Universal Robots PolyScope program: Programa_UR5_Gavetas.urp

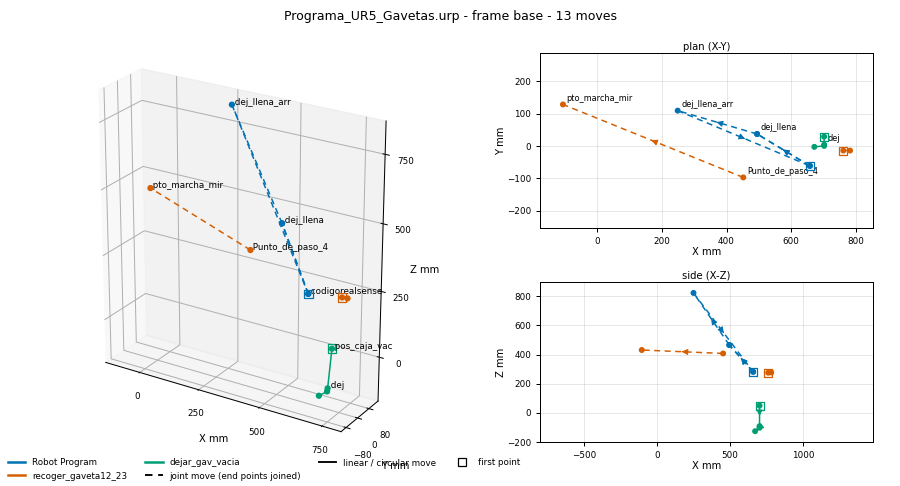
[picture p0: tool path of Programa_UR5_Gavetas.urp in frame base, 13 of 26 moves have a stored position in this frame; points joined in program order, loops and branches not executed]
Program Einnek_Planta240614 (installation=einnek directory=/programs/usbdisk/ur_mir createdIn=5.12.1.1101497 lastSavedIn=5.12.1.1101497 robotSerialNumber=20225590038)
Calibrated DH parameters: a=[0.000213, -0.400573, -0.367685, -0.000006, 0.000089, 0]; d=[0.162722, -86.393777, 65.991912, 20.535232, 0.099742, 0.099568]; alpha=[1.570328, 0.001648, 0.006729, 1.570321, -1.569293, 0]; deltaTheta=[0, -0.341442, -0.015889, 0.357341, 0.000001, 0]
InitVariablesNode variables(variable(name=ETAPA, expression=0), variable(name=IZQ_DER, expression=0), variable(name=LLENA_VACIA, expression=0), variable(name=Num_progr, expression=0), variable(name=pos_z, expression=0))
BeforeStart
  SuppressedNode
    Num_progr := 10   [initializeExpression=0]
  Folder Lectura posiciones
    URCap Read MiR register (MiRintegration, Mobile Industrial Robots APs) dataModel(register=Pos X, Variable(key=selectedVar, variable(name=pos_x, initializeExpression=0)))
    URCap Read MiR register (MiRintegration, Mobile Industrial Robots APs) dataModel(register=Pos Y, Variable(key=selectedVar, variable(name=pos_y, initializeExpression=0)))
    URCap Read MiR register (MiRintegration, Mobile Industrial Robots APs) dataModel(register=Pos Z, Variable(key=selectedVar, variable(name=pos_z, initializeExpression=0)))
    URCap Read MiR register (MiRintegration, Mobile Industrial Robots APs) dataModel(register=Rot X, Variable(key=selectedVar, variable(name=rot_x, initializeExpression=0)))
    URCap Read MiR register (MiRintegration, Mobile Industrial Robots APs) dataModel(register=Rot Y, Variable(key=selectedVar, variable(name=rot_y, initializeExpression=0)))
    URCap Read MiR register (MiRintegration, Mobile Industrial Robots APs) dataModel(register=Rot Z, Variable(key=selectedVar, variable(name=rot_z, initializeExpression=0)))
    URCap Read MiR register (MiRintegration, Mobile Industrial Robots APs) dataModel(register=IZQ_DER, Variable(key=selectedVar, variable(name=IZQ_DER, initializeExpression=0)))
    URCap Read MiR register (MiRintegration, Mobile Industrial Robots APs) dataModel(register=Altura_gaveta, Variable(key=selectedVar, variable(name=AbaArr)))
    SuppressedNode
      pos_caja := p[pos_x,pos_y,pos_z,rot_x,rot_y,rot_z]
    pos_caja := p[pos_x,pos_y,pos_z+0.12*AbaArr,rot_x,rot_y,rot_z]
  SuppressedNode
    AbaArr := 0
  SuppressedNode
    pos_caja := p[0,0,0,0,0,0]
Robot Program (runOnlyOnce=false)
  SafeHome (positionOptionType=SPEED_AND_ACCELERATION speed=1.047198 acceleration=1.396263 nextMotionTime=2)
  URCap Read MiR register (MiRintegration, Mobile Industrial Robots APs) dataModel(register=VACIA0_LLENA1, Variable(key=selectedVar, variable(name=LLENA_VACIA, initializeExpression=0)))
  If LLENA_VACIA≟1
    Folder PROGRAMA GAVETA LLENA
      URCap Read MiR register (MiRintegration, Mobile Industrial Robots APs) dataModel(register=ETAPAS, Variable(key=selectedVar, variable(name=ETAPA, initializeExpression=0)))
      Loop While (checkContinuously=false) expression=ETAPA≠101
        URCap Read MiR register (MiRintegration, Mobile Industrial Robots APs) dataModel(register=ETAPAS, Variable(key=selectedVar, variable=ETAPA))
        Wait Sleep waitTime=3
        Script: sync()
      MoveJ speed 60 deg/s, acceleration 80 deg/s^2 (useActiveTCP=true) feature=Base
        Waypoint codigorealsense: TCP in base x=657.88 y=-61.539 z=282.139 mm, rx=2.1337 ry=-2.1191 rz=-0.1759 rad; joints [160.264, -77.43, 101.576, -104.858, -93.53, -19.909] deg; TCP offset x=0 y=-115.54 z=0 mm, rx=0 ry=0 rz=0 rad
      Loop While (checkContinuously=false) expression=ETAPA≠103
        URCap Read MiR register (MiRintegration, Mobile Industrial Robots APs) dataModel(register=ETAPAS, Variable(key=selectedVar, variable=ETAPA))
        Wait Sleep waitTime=3
        Script: sync()
      Wait Sleep waitTime=1
      URCap Read MiR register (MiRintegration, Mobile Industrial Robots APs) dataModel(register=Pos_X_recogida, Variable(key=selectedVar, variable(name=PosXRecogida, initializeExpression=0)))
      Call recoger_gaveta12_23
      URCap Write MiR register (MiRintegration, Mobile Industrial Robots APs) dataModel(value=104, register=ETAPAS)
      URCap Read MiR register (MiRintegration, Mobile Industrial Robots APs) dataModel(register=ETAPAS, Variable(key=selectedVar, variable=ETAPA))
      Loop While (checkContinuously=false) expression=ETAPA≠106
        URCap Read MiR register (MiRintegration, Mobile Industrial Robots APs) dataModel(register=ETAPAS, Variable(key=selectedVar, variable=ETAPA))
        Wait Sleep waitTime=3
        Script: sync()
      Wait Condition expression=ETAPA≟106
      Folder Lectura posiciones
        URCap Read MiR register (MiRintegration, Mobile Industrial Robots APs) dataModel(register=Pos X, Variable(key=selectedVar, variable=pos_x))
        URCap Read MiR register (MiRintegration, Mobile Industrial Robots APs) dataModel(register=Pos Y, Variable(key=selectedVar, variable=pos_y))
        URCap Read MiR register (MiRintegration, Mobile Industrial Robots APs) dataModel(register=Pos Z, Variable(key=selectedVar, variable=pos_z))
        URCap Read MiR register (MiRintegration, Mobile Industrial Robots APs) dataModel(register=Rot X, Variable(key=selectedVar, variable=rot_x))
        URCap Read MiR register (MiRintegration, Mobile Industrial Robots APs) dataModel(register=Rot Y, Variable(key=selectedVar, variable=rot_y))
        URCap Read MiR register (MiRintegration, Mobile Industrial Robots APs) dataModel(register=Rot Z, Variable(key=selectedVar, variable=rot_z))
        URCap Read MiR register (MiRintegration, Mobile Industrial Robots APs) dataModel(register=IZQ_DER, Variable(key=selectedVar, variable=IZQ_DER))
        URCap Read MiR register (MiRintegration, Mobile Industrial Robots APs) dataModel(register=Altura_gaveta, Variable(key=selectedVar, variable=AbaArr))
        SuppressedNode
          pos_caja := p[pos_x,pos_y,pos_z,rot_x,rot_y,rot_z]
        SuppressedNode
          AbaArr := 0
        pos_caja := p[pos_x,pos_y,pos_z+0.12*AbaArr,rot_x,rot_y,rot_z]
      URCap Write MiR register (MiRintegration, Mobile Industrial Robots APs) dataModel(value=107, register=ETAPAS)
      If pos_z≤0.6
        MoveJ speed 60 deg/s, acceleration 80 deg/s^2 (useActiveTCP=true) feature=Base
          Waypoint dej_llena: motionParameters(jointSpeed=1.047198 jointAcceleration=0.436332 cartesianSpeed=0.25 cartesianAcceleration=1.2 blendRadius=0.05); TCP in base x=494.444 y=37.151 z=465.918 mm, rx=-2.1193 ry=2.1657 rz=-0.1543 rad; joints [165.601, -108.768, 117.243, -106.569, -87.444, -13.084] deg; TCP offset x=1.251 y=-112.953 z=-27.309 mm, rx=0 ry=0 rz=0 rad
      Else 
        MoveJ speed 60 deg/s, acceleration 80 deg/s^2 (useActiveTCP=true) feature=Base
          Waypoint dej_llena_arr: motionParameters(jointSpeed=1.047198 jointAcceleration=0.436332 cartesianSpeed=0.25 cartesianAcceleration=1.2 blendRadius=0.05); TCP in base x=248.72 y=109.415 z=823.024 mm, rx=-2.2887 ry=2.1434 rz=-0.0254 rad; joints [166.2, -111.162, 44.661, -24.388, -90.221, -17.987] deg; TCP offset x=0 y=-115.54 z=0 mm, rx=0 ry=0 rz=0 rad
      URCap Read MiR register (MiRintegration, Mobile Industrial Robots APs) dataModel(register=IZQ_DER, Variable(key=selectedVar, variable=IZQ_DER))
      If IZQ_DER≟1
        Call dejar_gav_der
      ElseIf IZQ_DER≟0
        Call dejar_gav_izq
      Else 
        Popup Message (haltProgram=false message=lado no asociado a codigo inputType=Text)
      URCap Write MiR register (MiRintegration, Mobile Industrial Robots APs) dataModel(value=108, register=ETAPAS)
      SafeHome (positionOptionType=SPEED_AND_ACCELERATION speed=1.047198 acceleration=1.396263 nextMotionTime=2)
  ElseIf LLENA_VACIA≟0
    Folder PROGRAMA GAVETA VACIA
      URCap Read MiR register (MiRintegration, Mobile Industrial Robots APs) dataModel(register=ETAPAS, Variable(key=selectedVar, variable=ETAPA))
      Loop While (checkContinuously=false) expression=ETAPA≠201
        URCap Read MiR register (MiRintegration, Mobile Industrial Robots APs) dataModel(register=ETAPAS, Variable(key=selectedVar, variable=ETAPA))
        Wait Sleep waitTime=3
        Script: sync()
      MoveJ speed 60 deg/s, acceleration 80 deg/s^2 (useActiveTCP=true) feature=Base
        Waypoint codigorealsense: TCP in base x=657.88 y=-61.539 z=282.139 mm, rx=2.1337 ry=-2.1191 rz=-0.1759 rad; joints [160.264, -77.43, 101.576, -104.858, -93.53, -19.909] deg
      Loop While (checkContinuously=false) expression=ETAPA≠203
        URCap Read MiR register (MiRintegration, Mobile Industrial Robots APs) dataModel(register=ETAPAS, Variable(key=selectedVar, variable=ETAPA))
        Wait Sleep waitTime=3
        Script: sync()
      Wait Condition expression=ETAPA≟203
      URCap Read MiR register (MiRintegration, Mobile Industrial Robots APs) dataModel(register=Pos_X_recogida, Variable(key=selectedVar, variable=PosXRecogida))
      Call recoger_gaveta12_23
      URCap Write MiR register (MiRintegration, Mobile Industrial Robots APs) dataModel(value=204, register=ETAPAS)
      SuppressedNode
        Folder Lectura posiciones
          URCap Read MiR register (MiRintegration, Mobile Industrial Robots APs) dataModel(register=Pos X, Variable(key=selectedVar, variable=pos_x))
          URCap Read MiR register (MiRintegration, Mobile Industrial Robots APs) dataModel(register=Pos Y, Variable(key=selectedVar, variable=pos_y))
          URCap Read MiR register (MiRintegration, Mobile Industrial Robots APs) dataModel(register=Pos Z, Variable(key=selectedVar, variable=pos_z))
          URCap Read MiR register (MiRintegration, Mobile Industrial Robots APs) dataModel(register=Rot X, Variable(key=selectedVar, variable=rot_x))
          URCap Read MiR register (MiRintegration, Mobile Industrial Robots APs) dataModel(register=Rot Y, Variable(key=selectedVar, variable=rot_y))
          URCap Read MiR register (MiRintegration, Mobile Industrial Robots APs) dataModel(register=Rot Z, Variable(key=selectedVar, variable=rot_z))
          URCap Read MiR register (MiRintegration, Mobile Industrial Robots APs) dataModel(register=IZQ_DER, Variable(key=selectedVar, variable=IZQ_DER))
          URCap Read MiR register (MiRintegration, Mobile Industrial Robots APs) dataModel(register=Altura_gaveta, Variable(key=selectedVar, variable=AbaArr))
          SuppressedNode
            pos_caja := p[pos_x,pos_y,pos_z,rot_x,rot_y,rot_z]
          SuppressedNode
            AbaArr := 0
          pos_caja := p[pos_x,pos_y,pos_z+0.12*AbaArr,rot_x,rot_y,rot_z]
      URCap Read MiR register (MiRintegration, Mobile Industrial Robots APs) dataModel(register=ETAPAS, Variable(key=selectedVar, variable=ETAPA))
      Loop While (checkContinuously=false) expression=ETAPA≠206
        URCap Read MiR register (MiRintegration, Mobile Industrial Robots APs) dataModel(register=ETAPAS, Variable(key=selectedVar, variable=ETAPA))
        Wait Sleep waitTime=3
        Script: sync()
      Wait Condition expression=ETAPA≟206
      URCap Write MiR register (MiRintegration, Mobile Industrial Robots APs) dataModel(value=207, register=ETAPAS)
      MoveJ speed 60 deg/s, acceleration 80 deg/s^2 (useActiveTCP=true) feature=Base
        Waypoint dej_gaveta_vac: TCP in base x=494.439 y=37.149 z=465.919 mm, rx=-2.1192 ry=2.1657 rz=-0.1543 rad; joints [165.136, -110.276, 114.29, -102.089, -87.384, -13.573] deg
      Call dejar_gav_vacia
      URCap Write MiR register (MiRintegration, Mobile Industrial Robots APs) dataModel(value=208, register=ETAPAS)
      SuppressedNode
        Wait Sleep waitTime=2
      SafeHome (positionOptionType=SPEED_AND_ACCELERATION speed=1.047198 acceleration=1.396263 nextMotionTime=2)
  ''
SubProgram -> recoger_gaveta12_23
SubProgram -> dejar_gav_izq
SubProgram -> dejar_gav_der
SubProgram -> dejar_gav_vacia
SuppressedNode
  Thread SubTarea_2 (runOnlyOnce=false)
    Script: socket_open("172.17.142.17",9000,"nodesocket")
    Script: socket_send_string(Num_progr,"nodesocket")
    Script: socket_close(socket_name="nodesocket")
SuppressedNode
  Thread SubTarea_1 (runOnlyOnce=false)
    URCap Read MiR register (MiRintegration, Mobile Industrial Robots APs) dataModel(register=ETAPAS, Variable(key=selectedVar, variable=ETAPA))
    Wait Sleep waitTime=1
    Script: sync()
SubProgram recoger_gaveta12_23 (keepSynchronizedWithDisk=false) programFile=/programs/ur_mir/recoger_gaveta12_23.urp
  MoveJ speed 60 deg/s, acceleration 80 deg/s^2 (useActiveTCP=true) feature=Base
    SuppressedNode
      Waypoint aprox_cogida: motionParameters(blendRadius=0.1); TCP in base x=598.101 y=11.394 z=33.528 mm, rx=-2.211 ry=2.1579 rz=-0.0851 rad; joints [165.134, -47.414, 126.392, -173.083, -88.815, -15.941] deg; TCP offset x=1.251 y=-112.953 z=-27.309 mm, rx=0 ry=0 rz=0 rad
    Waypoint recoger_gaveta: TCP in base x=761.406 y=-14.095 z=275.699 mm, rx=1.8647 ry=-1.861 rz=-0.6084 rad; joints [168.429, -55.339, 59.645, -58.808, -96.427, -9.91] deg; TCP offset x=0 y=-115.54 z=0 mm, rx=0 ry=0 rz=0 rad
  MoveL speed 250 mm/s, acceleration 1200 mm/s^2 (useActiveTCP=true) feature=Base
    Waypoint giro_touch: TCP in base x=782.119 y=-14.094 z=277.498 mm, rx=1.8647 ry=-1.861 rz=-0.6084 rad; joints [168.753, -51.968, 53.839, -56.343, -96.245, -9.657] deg
    MoveDirectionNode (selectedDirection=YPlus toolParams=0.025, 0.025) feature=Base
      Until TOOL_CONTACT_DETECTION (allowActions=false retraction=0.032 decelerationAcceleration=3 decelerationAngularAcceleration=34.906585)
      Until DISTANCE (allowActions=false deceleration=3 distanceNodeType=STOP) Distance=0.05; motionParameters(blendRadius=0)
    SuppressedNode
      Waypoint Punto_de_paso_2: TCP in base x=694.647 y=11.986 z=-102.063 mm, rx=1.5084 ry=-1.4533 rz=-0.9716 rad; joints [170.954, -28.236, 63.804, -58.084, -100.483, -4.371] deg
    SuppressedNode
      Halt
    MoveDirectionNode (selectedDirection=ZMinus toolParams=0.09, 1.2) feature=Joint_6_name
      Until TOOL_CONTACT_DETECTION (allowActions=false retraction=0.003 decelerationAcceleration=3 decelerationAngularAcceleration=34.906585)
      Until DISTANCE (allowActions=false deceleration=3 distanceNodeType=STOP) Distance=0.05; motionParameters(blendRadius=0)
    SuppressedNode
      MoveDirectionNode (selectedDirection=YPlus toolParams=0.09, 1.2) feature=Joint_6_name
        Until TOOL_CONTACT_DETECTION (allowActions=false retraction=0.001 decelerationAcceleration=3 decelerationAngularAcceleration=34.906585)
        Until DISTANCE (allowActions=false deceleration=3 distanceNodeType=STOP) Distance=0.05; motionParameters(blendRadius=0)
    MoveDirectionNode (selectedDirection=ZPlus toolParams=0.09, 1.2) feature=Base
      Until DISTANCE (allowActions=false deceleration=3 distanceNodeType=STOP) Distance=0.015; motionParameters(blendRadius=0)
    MoveL speed 250 mm/s, acceleration 1200 mm/s^2 (useActiveTCP=true) feature=Base
      Waypoint Punto_de_paso_3 (Relative): relativeFromPosition TCP in base x=691.72 y=18.401 z=-93.097 mm, rx=1.7603 ry=-1.7129 rz=-0.7082 rad; joints [170.664, -37.497, 85.202, -92.184, -98.673, -7.28] deg; TCP in base x=691.746 y=18.409 z=-93.092 mm, rx=1.9813 ry=-1.9435 rz=-0.403 rad; joints [169.815, -38.827, 99.063, -125.596, -96.241, -9.795] deg
    SuppressedNode
      Halt
    MoveDirectionNode (selectedDirection=ZPlus toolParams=0.09, 1.2) feature=Base
      Until DISTANCE (allowActions=false deceleration=3 distanceNodeType=STOP) Distance=0.05; motionParameters(blendRadius=0)
    MoveDirectionNode (selectedDirection=XMinus toolParams=0.09, 1.2) feature=Base
      Until DISTANCE (allowActions=false deceleration=3 distanceNodeType=STOP) Distance=0.01; motionParameters(blendRadius=0)
    SuppressedNode
      MoveDirectionNode (selectedDirection=XMinus toolParams=0.09, 1.2) feature=Base
        Until DISTANCE (allowActions=false deceleration=3 distanceNodeType=STOP) Distance=0.02; motionParameters(blendRadius=0)
    MoveL speed 250 mm/s, acceleration 1200 mm/s^2 (useActiveTCP=true) feature=Base
      Waypoint Punto_de_paso_4: motionParameters(blendRadius=0.1); TCP in base x=451.784 y=-97.223 z=407.756 mm, rx=-2.309 ry=2.1043 rz=0.1234 rad; joints [140.02, -111.366, 116.944, -91.005, -88.68, -45.499] deg
    SuppressedNode
      Waypoint giro_recogida (Relative): relativeFromPosition TCP in base x=707.318 y=18.52 z=-67.699 mm, rx=1.7336 ry=-1.7482 rz=-0.7236 rad; joints [170.916, -38.446, 81.943, -87.741, -97.043, -5.687] deg; TCP in base x=707.329 y=18.501 z=-67.678 mm, rx=-2.1827 ry=2.1799 rz=-0.1282 rad; joints [168.831, -32.029, 105.931, -169.497, -89.831, -10.959] deg
    SuppressedNode
      Halt
    SuppressedNode
      Waypoint subir_gavetaGir (Relative): relativeFromPosition TCP in base x=707.285 y=18.514 z=-67.717 mm, rx=-2.1827 ry=2.1799 rz=-0.1281 rad; joints [168.832, -32.029, 105.937, -169.496, -89.832, -10.958] deg; TCP in base x=534.855 y=18.524 z=-57.903 mm, rx=-2.1828 ry=2.1799 rz=-0.1282 rad; joints [163.928, -35.397, 133.647, -193.829, -89.506, -15.792] deg
    SuppressedNode
      Waypoint subida_gaveta (Relative): relativeFromPosition TCP in base x=731.204 y=-29.67 z=-62.84 mm, rx=2.1982 ry=-2.1997 rz=-0.1751 rad; joints [164.771, -32.645, 99.189, -150.105, -87.821, -15.098] deg; TCP offset x=1.251 y=-112.953 z=-27.309 mm, rx=0 ry=0 rz=0 rad; TCP in base x=731.202 y=-29.694 z=4.567 mm, rx=2.1981 ry=-2.1998 rz=-0.1751 rad; joints [164.777, -40.93, 101.485, -144.115, -87.809, -15.127] deg
    SuppressedNode
      Waypoint Punto_de_paso_1: motionParameters(blendRadius=0.05); TCP in base x=219.403 y=-208.448 z=635.733 mm, rx=-2.1267 ry=2.2581 rz=0.1182 rad; joints [83.053, -122.255, 87.405, -50.635, -91.894, -93.79] deg; TCP offset x=0 y=-115.54 z=0 mm, rx=0 ry=0 rz=0 rad
    SuppressedNode
      Waypoint Punto_de_paso_6: TCP in base x=246.18 y=-55.944 z=631.487 mm, rx=2.9564 ry=-0.8995 rz=-0.1048 rad; joints [108.981, -122.04, 88.698, -56.624, -94.687, -127.511] deg
  MoveJ speed 60 deg/s, acceleration 80 deg/s^2 (useActiveTCP=true) feature=Base
    Waypoint pto_marcha_mir: TCP in base x=-106.254 y=128.566 z=431.48 mm, rx=-2.1073 ry=2.1634 rz=-0.1712 rad; joints [179.689, -190.41, 113.522, -22.341, -90.026, 0.871] deg; TCP offset x=1.251 y=-112.953 z=-27.309 mm, rx=0 ry=0 rz=0 rad
SubProgram dejar_gav_der (keepSynchronizedWithDisk=false) programFile=/programs/ur_mir/dejar_gav_der.urp
  SuppressedNode
    URCap Read MiR register (MiRintegration, Mobile Industrial Robots APs) dataModel(register=Altura_gaveta, Variable(key=selectedVar, variable=AbaArr))
  SuppressedNode
    If AbaArr≟0 removedSiblings(If(type=Else checkContinuously=false, children(Move(motionType=MoveJ speed=1.047198 acceleration=1.396263 useActiveTCP=true positionType=CartesianPose, feature=Base, children(Waypoint(type=Fixed name=AproxGavDchArr, position(JointAngles=[2.670034, -0.950152, 2.176509, -2.920692, -1.767392, 1.068185], TCPOffset=[0.001251, -0.112953, -0.027309, 0, 0, 0]), BaseToFeature=[0, 0, 0, 0, 0, 0]))))))
      MoveJ speed 60 deg/s, acceleration 80 deg/s^2 (useActiveTCP=true) feature=Base
        Waypoint AproxGavDchAba: TCP in base x=488.698 y=-225.557 z=-13.138 mm, rx=-0.0362 ry=3.1031 rz=-0.3674 rad; joints [152.967, -35.552, 120.582, -182.097, -101.325, 61.248] deg
  SuppressedNode
    MoveJ speed 60 deg/s, acceleration 80 deg/s^2 (useActiveTCP=true) feature=Base
      Waypoint AproxGavDchAba: TCP in base x=488.698 y=-225.557 z=-13.138 mm, rx=-0.0362 ry=3.1031 rz=-0.3674 rad; joints [152.967, -35.552, 120.582, -182.097, -101.325, 61.248] deg
  MoveJ speed 60 deg/s, acceleration 80 deg/s^2 (useActiveTCP=true) feature=Base
    SuppressedNode
      Waypoint AproxGavDchAba: TCP in base x=488.698 y=-225.557 z=-13.138 mm, rx=-0.0362 ry=3.1031 rz=-0.3674 rad; joints [152.967, -35.552, 120.582, -182.097, -101.325, 61.248] deg
    SuppressedNode
      pos_caja := p[pos_x,pos_y,pos_z+0.12*AbaArr,rot_x,rot_y,rot_z]
    Waypoint Punto_de_paso (Variable): variable=pos_caja
    SuppressedNode
      Waypoint prubapaso: TCP in base x=488.708 y=-165.163 z=285.307 mm, rx=-0.0365 ry=3.1033 rz=-0.367 rad; joints [160.674, -82.48, 119.78, -132.784, -102.015, 68.819] deg; TCP offset x=0 y=-115.54 z=0 mm, rx=0 ry=0 rz=0 rad
  MoveL speed 250 mm/s, acceleration 1200 mm/s^2 (useActiveTCP=true) feature=Base
    SuppressedNode
      Waypoint dejar_1_der (Relative): relativeFromPosition TCP in base x=488.682 y=-225.564 z=-13.143 mm, rx=-0.0378 ry=3.122 rz=-0.1648 rad; joints [153.197, -43.312, 123.432, -173.572, -94.765, 61.953] deg; TCP offset x=0 y=-120 z=0 mm, rx=0 ry=0 rz=0 rad; TCP in base x=488.681 y=-454.462 z=-13.153 mm, rx=-0.0378 ry=3.122 rz=-0.1648 rad; joints [133.003, -39.282, 108.38, -164.05, -93.168, 41.729] deg
    Waypoint DejDch1 (Relative): relativeFromPosition TCP in base x=488.681 y=-225.56 z=-13.158 mm, rx=-0.0361 ry=3.1032 rz=-0.3674 rad; joints [152.966, -35.55, 120.583, -182.096, -101.326, 61.249] deg; TCP offset x=1.251 y=-112.953 z=-27.309 mm, rx=0 ry=0 rz=0 rad; TCP in base x=488.693 y=-563.866 z=-13.137 mm, rx=-0.0362 ry=3.1032 rz=-0.3674 rad; joints [126.331, -28.504, 92.905, -165.864, -96.784, 34.575] deg
    Waypoint DejDch2 (Relative): relativeFromPosition TCP in base x=488.69 y=-541.838 z=-13.158 mm, rx=-0.0362 ry=3.1032 rz=-0.3674 rad; joints [127.527, -29.368, 95.66, -167.604, -97.034, 35.762] deg; TCP in base x=488.693 y=-541.863 z=-91.249 mm, rx=-0.0361 ry=3.1031 rz=-0.3675 rad; joints [127.521, -19.53, 90.54, -172.324, -97.051, 35.787] deg
    Waypoint GiroDch1 (Relative): relativeFromPosition TCP in base x=488.691 y=-541.86 z=-91.249 mm, rx=-0.0361 ry=3.1031 rz=-0.3675 rad; joints [127.521, -19.53, 90.541, -172.325, -97.05, 35.788] deg; TCP in base x=488.688 y=-541.833 z=-91.278 mm, rx=-0.0399 ry=3.1253 rz=0.147 rad; joints [126.395, -27.095, 92.667, -151.538, -85.956, 35.006] deg
    Waypoint GiroDch2 (Relative): relativeFromPosition TCP in base x=488.699 y=-541.846 z=-91.258 mm, rx=-0.04 ry=3.1253 rz=0.147 rad; joints [126.395, -27.095, 92.665, -151.539, -85.956, 35.004] deg; TCP in base x=488.686 y=-541.847 z=-137.943 mm, rx=-0.04 ry=3.1253 rz=0.147 rad; joints [126.39, -21.298, 89.659, -154.33, -85.963, 35.02] deg
  SuppressedNode
    MoveJ speed 60 deg/s, acceleration 80 deg/s^2 (useActiveTCP=true) feature=Base
      Waypoint AproxGavDchAba: TCP in base x=488.698 y=-225.557 z=-13.138 mm, rx=-0.0362 ry=3.1031 rz=-0.3674 rad; joints [152.967, -35.552, 120.582, -182.097, -101.325, 61.248] deg
  MoveJ speed 60 deg/s, acceleration 80 deg/s^2 (useActiveTCP=true) feature=Base
    SuppressedNode
      pos_caja := p[pos_x,pos_y,pos_z+0.12*AbaArr,rot_x,rot_y,rot_z]
    Waypoint Punto_de_paso (Variable): variable=pos_caja
SubProgram dejar_gav_izq (keepSynchronizedWithDisk=false) programFile=/programs/ur_mir/dejar_gav_izq.urp
  SuppressedNode
    URCap Read MiR register (MiRintegration, Mobile Industrial Robots APs) dataModel(register=Altura_gaveta, Variable(key=selectedVar, variable=AbaArr))
  MoveJ speed 60 deg/s, acceleration 80 deg/s^2 (useActiveTCP=true) feature=Base
    SuppressedNode
      Waypoint Punto_de_paso_7: TCP in base x=473.654 y=206.93 z=361.7 mm, rx=-2.9615 ry=-0.0391 rz=0.0153 rad; joints [173.149, -89.887, 111.485, -109.529, -79.547, -98.622] deg; TCP offset x=0 y=-115.54 z=0 mm, rx=0 ry=0 rz=0 rad
    SuppressedNode
      pos_caja := p[pos_x,pos_y,pos_z+0.12*AbaArr,rot_x,rot_y,rot_z]
    Waypoint Punto_de_paso (Variable): variable=pos_caja
  SuppressedNode
    If AbaArr≟0 removedSiblings(If(type=Else checkContinuously=false, children(Move(motionType=MoveJ speed=1.047198 acceleration=1.396263 useActiveTCP=true positionType=CartesianPose, feature=Base, children(SuppressedNode(suppressedNode(type=Fixed name=AproxGavIzqArr, position(JointAngles=[3.097953, -1.201858, 2.1771, -2.524636, -1.386806, -1.640636], TCPOffset=[0, -0.12, 0, 0, 0, 0]), BaseToFeature=[0, 0, 0, 0, 0, 0])), Assignment(valueSource=Expression, variable=pos_caja, expression=p[pos_x,pos_y,pos_z+0.12*AbaArr,rot_x,rot_y,rot_z]), Waypoint(type=Variable name=Punto_de_paso, variable=pos_caja))))))
      MoveJ speed 60 deg/s, acceleration 80 deg/s^2 (useActiveTCP=true) feature=Base
        SuppressedNode
          Waypoint AproxGavIzqAba: motionParameters(jointSpeed=1.047198 jointAcceleration=1.396263 cartesianSpeed=0.25 cartesianAcceleration=1.2); TCP in base x=473.693 y=247.619 z=32.164 mm, rx=-2.9615 ry=-0.0396 rz=0.0148 rad; joints [177.472, -50.378, 125.236, -163.642, -79.516, -93.931] deg; TCP offset x=0 y=-120 z=0 mm, rx=0 ry=0 rz=0 rad
        pos_caja := p[pos_x,pos_y,pos_z+0.12*AbaArr,rot_x,rot_y,rot_z]
        Waypoint Punto_de_paso (Variable): variable=pos_caja
  MoveL speed 250 mm/s, acceleration 1200 mm/s^2 (useActiveTCP=true) feature=Base
    SuppressedNode
      Wait Sleep waitTime=10
    Waypoint DejIzq1 (Relative): relativeFromPosition TCP in base x=473.942 y=248.508 z=32.154 mm, rx=-2.9616 ry=-0.0396 rz=0.0147 rad; joints [177.582, -50.352, 125.164, -163.618, -79.518, -93.819] deg; TCP in base x=473.235 y=449.53 z=32.238 mm, rx=-2.9615 ry=-0.0388 rz=0.0157 rad; joints [200.308, -45.12, 111.189, -158.931, -79.821, -70.721] deg; TCP offset x=0 y=-115.54 z=0 mm, rx=0 ry=0 rz=0 rad
    SuppressedNode
      Wait Sleep waitTime=2
    Waypoint DejIzq2 (Relative): relativeFromPosition TCP in base x=172.294 y=448.618 z=823.075 mm, rx=-2.9615 ry=-0.0384 rz=0.0161 rad; joints [219.743, -91.555, 41.115, -45.456, -81.503, -51.733] deg; TCP in base x=172.302 y=448.619 z=784.377 mm, rx=-2.9614 ry=-0.0384 rz=0.016 rad; joints [219.742, -96.684, 53.878, -53.1, -81.468, -51.705] deg
    SuppressedNode
      Wait Sleep waitTime=2
    Waypoint giro1 (Relative): relativeFromPosition TCP in base x=172.309 y=448.628 z=784.379 mm, rx=-2.9614 ry=-0.0384 rz=0.016 rad; joints [219.743, -96.682, 53.876, -53.101, -81.469, -51.704] deg; TCP in base x=172.278 y=448.604 z=784.405 mm, rx=2.9588 ry=0.0406 rz=-0.0087 rad; joints [224.113, -81.149, 22.951, -24.313, -97.383, -47.416] deg
    Waypoint bajada (Relative): relativeFromPosition TCP in base x=473.001 y=450.05 z=-91.576 mm, rx=2.5221 ry=0.0321 rz=-0.0204 rad; joints [208.849, -39.203, 99.487, -130.759, -119.971, -57.168] deg; TCP in base x=472.992 y=450.061 z=-134.033 mm, rx=2.5222 ry=0.0321 rz=-0.0204 rad; joints [208.845, -34.077, 98.1, -134.485, -119.972, -57.146] deg
    Waypoint separar_izq (Relative): relativeFromPosition TCP in base x=473.012 y=450.08 z=-127.029 mm, rx=2.5222 ry=0.0321 rz=-0.0203 rad; joints [208.846, -34.931, 98.367, -133.903, -119.972, -57.149] deg; TCP in base x=472.989 y=402.403 z=-127.041 mm, rx=2.5222 ry=0.0321 rz=-0.0203 rad; joints [204.787, -36.279, 103.936, -140.41, -121.261, -61.597] deg
    SafeHome (positionOptionType=SPEED_AND_ACCELERATION speed=1.047198 acceleration=1.396263 nextMotionTime=2)
  SuppressedNode
    If AbaArr≟0 removedSiblings(If(type=Else checkContinuously=false, children(Move(motionType=MoveJ speed=1.047198 acceleration=1.396263 useActiveTCP=true positionType=CartesianPose, feature=Base, children(Waypoint(type=Fixed name=AproxGavIzqArr, position(JointAngles=[3.097953, -1.201858, 2.1771, -2.524636, -1.386806, -1.640636], TCPOffset=[0, -0.12, 0, 0, 0, 0]), BaseToFeature=[0, 0, 0, 0, 0, 0]))))))
      MoveJ speed 60 deg/s, acceleration 80 deg/s^2 (useActiveTCP=true) feature=Base
        Waypoint AproxGavIzqAba: TCP in base x=473.693 y=247.619 z=32.164 mm, rx=-2.9615 ry=-0.0396 rz=0.0148 rad; joints [177.472, -50.378, 125.236, -163.642, -79.516, -93.931] deg; TCP offset x=0 y=-120 z=0 mm, rx=0 ry=0 rz=0 rad
SubProgram dejar_gav_vacia (keepSynchronizedWithDisk=false) programFile=/programs/ur_mir/dejar_gav_izq.urp
  MoveJ speed 60 deg/s, acceleration 80 deg/s^2 (useActiveTCP=true) feature=Base
    Waypoint pos_caja_vac: TCP in base x=701.948 y=28.9 z=50.012 mm, rx=2.2531 ry=-2.1112 rz=-0.0933 rad; joints [169.178, -51.369, 107.951, -141.962, -90.371, -14.379] deg; TCP offset x=0 y=-115.54 z=0 mm, rx=0 ry=0 rz=0 rad
  SuppressedNode
    URCap Read MiR register (MiRintegration, Mobile Industrial Robots APs) dataModel(register=Altura_gaveta, Variable(key=selectedVar, variable=AbaArr))
  SuppressedNode
    MoveJ speed 60 deg/s, acceleration 80 deg/s^2 (useActiveTCP=true positionType=JointAngles) feature=Base
      SuppressedNode
        pos_caja := p[pos_x,pos_y,pos_z+0.12*AbaArr,rot_x,rot_y,rot_z]
      Waypoint Punto_de_paso (Variable): variable=pos_caja
  SuppressedNode
    If AbaArr≟0 removedSiblings(If(type=Else checkContinuously=false, children(Move(motionType=MoveJ speed=1.047198 acceleration=1.396263 useActiveTCP=true positionType=CartesianPose, feature=Base, children(SuppressedNode(suppressedNode(type=Fixed name=AproxGavIzqArr, position(JointAngles=[3.097953, -1.201858, 2.1771, -2.524636, -1.386806, -1.640636], TCPOffset=[0, -0.12, 0, 0, 0, 0]), BaseToFeature=[0, 0, 0, 0, 0, 0])), Assignment(valueSource=Expression, variable=pos_caja, expression=p[pos_x,pos_y,pos_z+0.12*AbaArr,rot_x,rot_y,rot_z]), Waypoint(type=Variable name=Punto_de_paso, variable=pos_caja))))))
      MoveJ speed 60 deg/s, acceleration 80 deg/s^2 (useActiveTCP=true) feature=Base
        SuppressedNode
          Waypoint AproxGavIzqAba: motionParameters(jointSpeed=1.047198 jointAcceleration=1.396263 cartesianSpeed=0.25 cartesianAcceleration=1.2); TCP in base x=473.693 y=247.619 z=32.164 mm, rx=-2.9615 ry=-0.0396 rz=0.0148 rad; joints [177.472, -50.378, 125.236, -163.642, -79.516, -93.931] deg; TCP offset x=0 y=-120 z=0 mm, rx=0 ry=0 rz=0 rad
        pos_caja := p[pos_x,pos_y,pos_z+0.12*AbaArr,rot_x,rot_y,rot_z]
        Waypoint Punto_de_paso (Variable): variable=pos_caja
  MoveL speed 250 mm/s, acceleration 1200 mm/s^2 (useActiveTCP=true) feature=Base
    SuppressedNode
      Waypoint DejIzq1 (Relative): relativeFromPosition TCP in base x=473.942 y=248.508 z=32.154 mm, rx=-2.9616 ry=-0.0396 rz=0.0147 rad; joints [177.582, -50.352, 125.164, -163.618, -79.518, -93.819] deg; TCP in base x=473.726 y=439.007 z=32.159 mm, rx=-2.9616 ry=-0.0395 rz=0.0148 rad; joints [199.269, -45.465, 112.121, -159.366, -79.787, -71.8] deg; TCP offset x=0 y=-115.54 z=0 mm, rx=0 ry=0 rz=0 rad
    Waypoint dej: TCP in base x=701.956 y=3.846 z=-91.587 mm, rx=2.1424 ry=-2.0081 rz=-0.3054 rad; joints [167.277, -36.909, 101.375, -138.643, -92.993, -15.839] deg
    SuppressedNode
      Waypoint DejIzq2 (Relative): relativeFromPosition TCP in base x=473.715 y=471.998 z=32.144 mm, rx=-2.9616 ry=-0.0395 rz=0.0148 rad; joints [202.002, -44.278, 109.282, -158.187, -79.922, -69.032] deg; TCP offset x=0 y=-120 z=0 mm, rx=0 ry=0 rz=0 rad; TCP in base x=701.917 y=28.921 z=-91.628 mm, rx=2.2531 ry=-2.111 rz=-0.0933 rad; joints [169.16, -33.426, 104.563, -156.512, -90.409, -14.313] deg; TCP offset x=0 y=-115.54 z=0 mm, rx=0 ry=0 rz=0 rad
    SuppressedNode
      Waypoint GiroIzq1 (Relative): relativeFromPosition TCP in base x=473.712 y=471.988 z=-91.739 mm, rx=-2.9616 ry=-0.0395 rz=0.0148 rad; joints [201.989, -27.775, 103.89, -169.306, -79.962, -68.983] deg; TCP offset x=0 y=-120 z=0 mm, rx=0 ry=0 rz=0 rad; TCP in base x=473.749 y=472.027 z=-91.694 mm, rx=3.0939 ry=0.0426 rz=-0.0105 rad; joints [203.914, -32.235, 104, -160.247, -92.066, -67.385] deg
    SuppressedNode
      Waypoint GiroIzq2 (Relative): relativeFromPosition TCP in base x=701.968 y=28.936 z=-73.837 mm, rx=2.1219 ry=-1.9863 rz=-0.3158 rad; joints [169.816, -39.377, 101.241, -134.579, -93.384, -13.293] deg; TCP offset x=0 y=-115.54 z=0 mm, rx=0 ry=0 rz=0 rad; TCP in base x=701.973 y=28.944 z=-99.982 mm, rx=1.7602 ry=-1.6414 rz=-0.8172 rad; joints [171.09, -34.68, 79.128, -84.349, -97.235, -9.59] deg
    Waypoint Punto_de_paso_5: TCP in base x=701.967 y=0.388 z=-101.909 mm, rx=1.8644 ry=-1.7486 rz=-0.7111 rad; joints [168.225, -36.53, 86.452, -98.833, -97.278, -12.707] deg
    Waypoint Punto_de_sal2: TCP in base x=671.644 y=-2.597 z=-125.704 mm, rx=1.8644 ry=-1.7486 rz=-0.711 rad; joints [167.399, -36.482, 92.116, -104.631, -97.816, -13.297] deg
  SuppressedNode
    If AbaArr≟0 removedSiblings(If(type=Else checkContinuously=false, children(Move(motionType=MoveJ speed=1.047198 acceleration=1.396263 useActiveTCP=true positionType=CartesianPose, feature=Base, children(Waypoint(type=Fixed name=AproxGavIzqArr, position(JointAngles=[3.097953, -1.201858, 2.1771, -2.524636, -1.386806, -1.640636], TCPOffset=[0, -0.12, 0, 0, 0, 0]), BaseToFeature=[0, 0, 0, 0, 0, 0]))))))
      MoveJ speed 60 deg/s, acceleration 80 deg/s^2 (useActiveTCP=true) feature=Base
        Waypoint AproxGavIzqAba: TCP in base x=473.693 y=247.619 z=32.164 mm, rx=-2.9615 ry=-0.0396 rz=0.0148 rad; joints [177.472, -50.378, 125.236, -163.642, -79.516, -93.931] deg; TCP offset x=0 y=-120 z=0 mm, rx=0 ry=0 rz=0 rad
  SuppressedNode
    MoveJ speed 60 deg/s, acceleration 80 deg/s^2 (useActiveTCP=true) feature=Base
      Waypoint pos_caja_vac: TCP in base x=701.948 y=28.9 z=50.012 mm, rx=2.2531 ry=-2.1112 rz=-0.0933 rad; joints [169.178, -51.369, 107.951, -141.962, -90.371, -14.379] deg; TCP offset x=0 y=-115.54 z=0 mm, rx=0 ry=0 rz=0 rad
